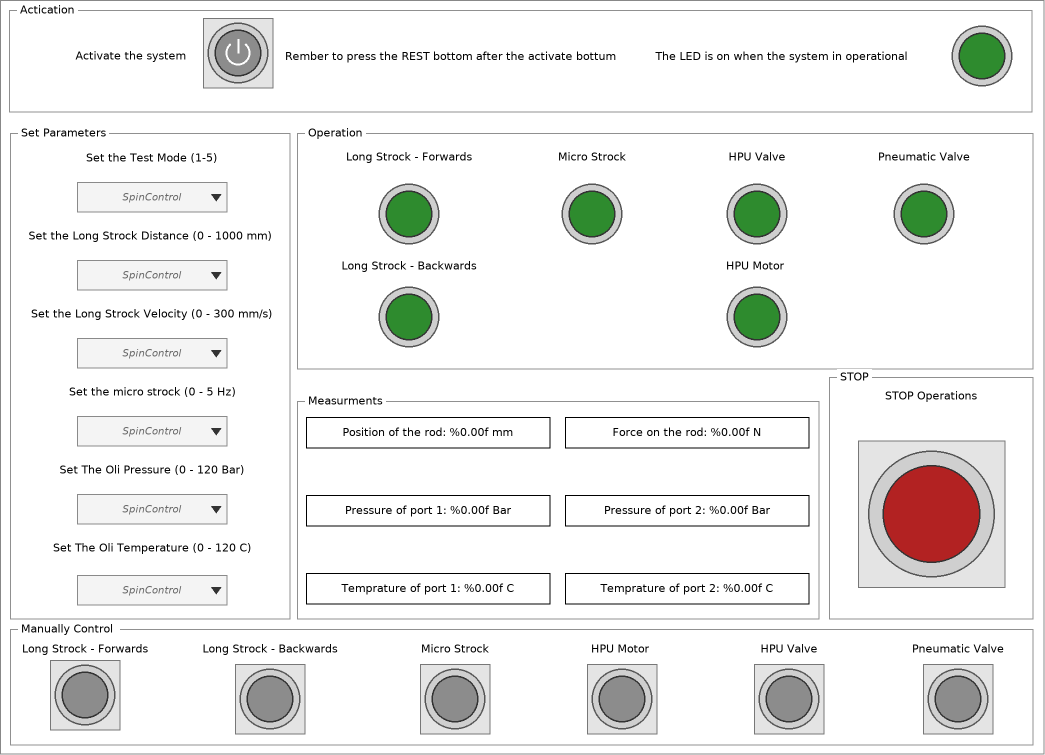
VISUALIZATION Visualization  // 1045x755
    GroupBox (9,2 1023x110), "Actication"
        Label (38,26 168x56), "Activate the system"
        Label (276,40 331x29), "Rember to press the REST bottom after the activate bottum"
        Lamp1 (938,19 70x70), variable: MAIN.fbSafetyBlock.bSystemIsUpAndRuning, style: Lamp-Lamp1-Green
        Label (607,40 331x29), "The LED is on when the system in operational"
        PowerSwitch (194,16 70x70), variable: MAIN.fbSafetyBlock.bHmiActivationBottom, behaviour: TOGGLE, style: Switch-PowerSwitch-Gray
    GroupBox (10,125 280x494), "Set Parameters"
        SpinControl (67,57 150x30), variable: MAIN.iTestMode
            OnMouseClick: write the text variable via Edit, min 0, max 5, format %i
        SpinControl (67,291 150x30), variable: MAIN.rMicroStrockAngularSpeedSet
            p1653691745: 0.1
            OnMouseClick: write the text variable via Edit, min 0, max 1000, format %r
        SpinControl (67,369 150x30), variable: MAIN.rOilPressureSet
            OnMouseClick: write the text variable via Edit, min 0, max 120, format %r
        SpinControl (67,450 150x30), variable: MAIN.rOilTemperatureSet
            OnMouseClick: write the text variable via Edit, min 0, max 120, format %r
        Label (67,18 150x30), "Set the Test Mode (1-5)"
        Label (50,252 185x30), "Set the micro strock (0 - 5 Hz)"
        Label (28,408 229x30), "Set The Oli Temperature (0 - 120 C)"
        Label (39,330 206x30), "Set The Oli Pressure (0 - 120 Bar)"
        SpinControl (67,135 150x30), variable: MAIN.rLongStrockDistanceSet
            OnMouseClick: write the text variable via Edit, min 0, max 1000, format %i
        Label (11,96 262x30), "Set the Long Strock Distance (0 - 1000 mm)"
        SpinControl (67,213 150x30), variable: MAIN.fbVfdBlock.rSet
            OnMouseClick: write the text variable via Edit, min 0, max 300, format %i
        Label (13,174 258x30), "Set the Long Strock Velocity (0 - 300 mm/s)"
    GroupBox (297,393 522x226), "Measurments"
        RoundedRectangle (9,180 244x31), "Temprature of port 1: %0.00f C", text variable: MAIN.rTemperatureReadable1
        RoundedRectangle (268,180 244x31), "Temprature of port 2: %0.00f C", text variable: MAIN.rTemperatureReadable2
        RoundedRectangle (9,102 244x31), "Pressure of port 1: %0.00f Bar", text variable: MAIN.rPerssureReadable1
        RoundedRectangle (268,102 244x31), "Pressure of port 2: %0.00f Bar", text variable: MAIN.rPerssureReadable2
        RoundedRectangle (268,24 244x31), "Force on the rod: %0.00f N", text variable: MAIN.rForceReadable
        RoundedRectangle (9,24 244x31), "Position of the rod: %0.00f mm", text variable: MAIN.rPositionReadable
    GroupBox (297,125 736x244), "Operation"
        Lamp1 (425,54 70x70), variable: MAIN.fbHpuBlock.bHpuValveControlRelayFive, style: Lamp-Lamp1-Green
        Lamp1 (425,157 70x70), variable: MAIN.fbHpuBlock.bHpuMotorControlRelayTwo, style: Lamp-Lamp1-Green
        Label (385,126 150x30), "HPU Motor"
        Label (385,17 150x30), "HPU Valve"
        Lamp1 (592,54 70x70), style: Lamp-Lamp1-Green
        Label (552,17 150x30), "Pneumatic Valve"
        Lamp1 (260,54 70x70), style: Lamp-Lamp1-Green
        Label (220,17 150x30), "Micro Strock"
        Lamp1 (77,54 70x70), style: Lamp-Lamp1-Green
        Label (37,17 150x30), "Long Strock - Forwards"
        Lamp1 (77,157 70x70), style: Lamp-Lamp1-Green
        Label (19,126 186x30), "Long Strock - Backwards"
    GroupBox (829,369 204x250), "STOP"
        Label (27,12 150x30), "STOP Operations"
        PushSwitchLed (29,63 147x164), variable: MAIN.bSTOP, behaviour: TOGGLE, style: Switch-PushSwitchLed-Red
    GroupBox (10,621 1023x124), "Manually Control"
        Label (0,13 150x30), "Long Strock - Forwards"
        Label (167,13 186x30), "Long Strock - Backwards"
        Label (370,13 150x30), "Micro Strock"
        Label (537,13 150x30), "HPU Motor"
        Label (704,13 150x30), "HPU Valve"
        Label (873,13 150x30), "Pneumatic Valve"
        PushSwitchLed (40,39 70x70), variable: MAIN.fbVfdBlock.bOnOffVfd1ControlRelaySeven, behaviour: TOGGLE, style: Switch-PushSwitchLed-Gray
        PushSwitchLed (225,43 70x70), behaviour: TAP, style: Switch-PushSwitchLed-Gray
        PushSwitchLed (410,43 70x70), behaviour: TAP, style: Switch-PushSwitchLed-Gray
        PushSwitchLed (577,43 70x70), variable: MAIN.fbHpuBlock.bHpuMotorControlRelayTwo, behaviour: TAP, style: Switch-PushSwitchLed-Gray
        PushSwitchLed (744,43 70x70), variable: MAIN.fbHpuBlock.bHpuValveControlRelayFive, behaviour: TOGGLE, style: Switch-PushSwitchLed-Gray
        PushSwitchLed (913,43 70x70), behaviour: TAP, style: Switch-PushSwitchLed-Gray
END_VISUALIZATION

(* stored: Version 1.1.0.1, ProductVersion 3.1.4024.16
   Visu Visualization: Id {b192a8e5-3a89-4284-8250-c99b5b63a344} *)
